FUNCTION_BLOCK FB_Estacion
VAR_INPUT
	// SFC-Flags
	SFCReset: BOOL;
	
	// Parámetros
	TpoEstabilidad: TIME := T#1000MS;
	UdsSolicitadas:UINT := 5;
	
END_VAR
VAR_OUTPUT
	// Parámetros
	CondicionInicial: BOOL;
	UdsPendientes: UINT;
	UdsRealizadas: BOOL;
	
	// Entradas comunes
	PulsadorEmergencia AT %I*: BOOL;
    SelectorManual AT %I*: BOOL;
    PulsadorMarcha AT %I*: BOOL;
    PulsadorParada AT %I*: BOOL := TRUE; // Contacto normalmente cerrado
    EstacionConectada AT %I*: BOOL := TRUE;
    DetectorPresion AT %I*: BOOL := TRUE;
	
	PalePresencia AT %I*: BOOL;
    PaleCodigoBit0 AT %I*: BOOL;
    PaleCodigoBit1 AT %I*: BOOL;
    PaleCodigoBit2 AT %I*: BOOL;
	
	// Entradas específicas
	DescargadorDetras AT %I*: BOOL;
	DescargadorDelante AT %I*: BOOL;
	VerticalArriba AT %I*: BOOL;
	VerticalAbajo AT %I*: BOOL;
	VerificadorArriba AT %I*: BOOL;
	VerificadorAbajo AT %I*: BOOL;
	DesplazadorDetras AT %I*: BOOL;
	AlimentadorDetras AT %I*: BOOL;
	AlimentadorDelante AT %I*: BOOL;
	VacioDescargador AT %I*: BOOL;
	PresenciaBaseAlimentador AT %I*:BOOL;
END_VAR
VAR
	// Bloques funcionales
	CLK: FB_Clock;
	// Salidas comunes
	DesconectaEstacion AT %Q*: BOOL;
    LamparaAlarma AT %Q*: BOOL;
    LamparaMarcha AT %Q*: BOOL;
	LamparaFaltaMaterial AT %Q*: BOOL;
    AvisadorSonoro AT %Q*: BOOL;

    CintaMotorActiva AT %Q*: BOOL;
    CintaMotorInvierte AT %Q*: BOOL;
    CintaRetenedorBaja AT %Q*: BOOL;
    CintaSeparadorSube AT %Q*: BOOL;
	
	// Salidas específicas
	DescargadorAtras AT %Q*: BOOL;
	DescargadorAdelante AT %Q*: BOOL;
	DescargadorBaja AT %Q*: BOOL;
	RechazadorAdelante AT %Q*: BOOL;
	VerificadorBaja AT %Q*: BOOL;
	DesplazadorAdelante AT %Q*: BOOL;
	AlimentadorAdelante AT %Q*: BOOL;
	EyectorSucciona AT %Q*: BOOL;
END_VAR

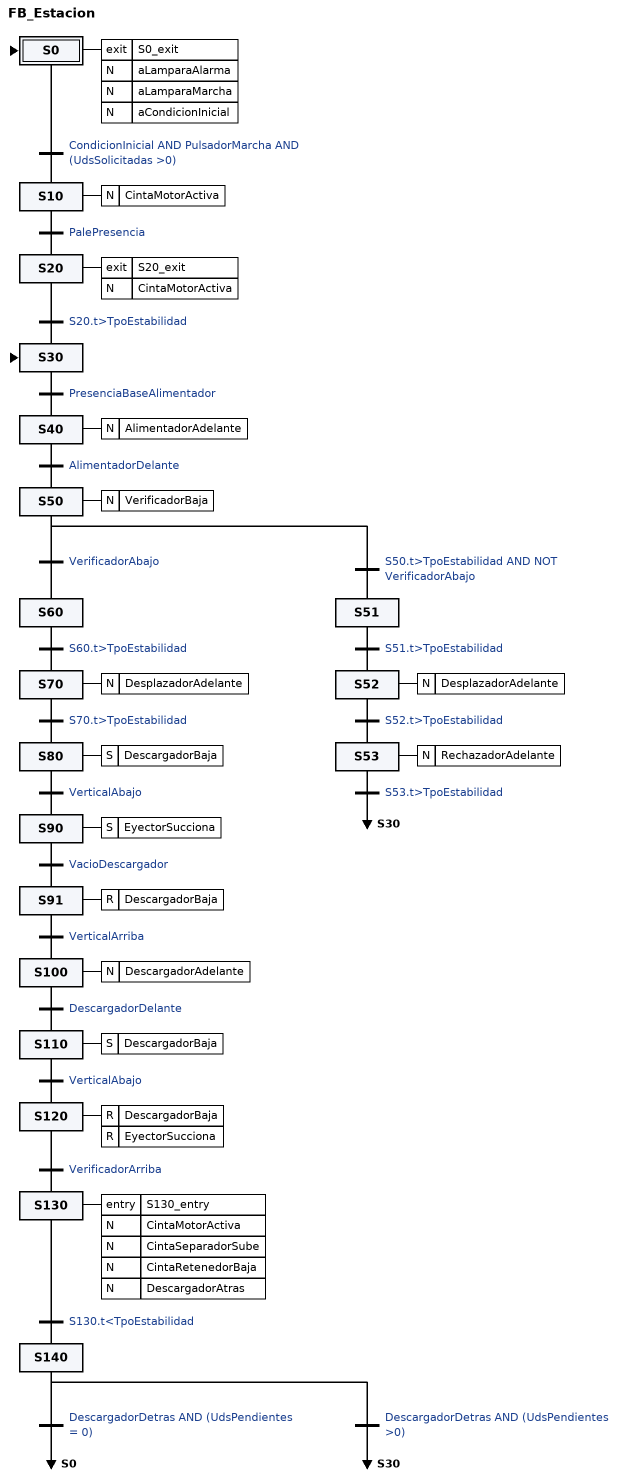
INITIAL_STEP S0:
    S0_exit(P0);  // exit action
    aLamparaAlarma(N);
    aLamparaMarcha(N);
    aCondicionInicial(N);
END_STEP
TRANSITION FROM S0 TO S10
    := CondicionInicial AND PulsadorMarcha AND (UdsSolicitadas >0);
END_TRANSITION
STEP S10:
    CintaMotorActiva(N);
END_STEP
TRANSITION FROM S10 TO S20
    := PalePresencia;
END_TRANSITION
STEP S20:
    S20_exit(P0);  // exit action
    CintaMotorActiva(N);
END_STEP
TRANSITION FROM S20 TO S30
    := S20.t>TpoEstabilidad;
END_TRANSITION
STEP S30:
END_STEP
TRANSITION FROM S30 TO S40
    := PresenciaBaseAlimentador;
END_TRANSITION
STEP S40:
    AlimentadorAdelante(N);
END_STEP
TRANSITION FROM S40 TO S50
    := AlimentadorDelante;
END_TRANSITION
STEP S50:
    VerificadorBaja(N);
END_STEP
TRANSITION FROM S50 TO S60
    := VerificadorAbajo;
END_TRANSITION
TRANSITION FROM S50 TO S51
    := S50.t>TpoEstabilidad AND NOT VerificadorAbajo;
END_TRANSITION
STEP S51:
END_STEP
TRANSITION FROM S51 TO S52
    := S51.t>TpoEstabilidad;
END_TRANSITION
STEP S52:
    DesplazadorAdelante(N);
END_STEP
TRANSITION FROM S52 TO S53
    := S52.t>TpoEstabilidad;
END_TRANSITION
STEP S53:
    RechazadorAdelante(N);
END_STEP
TRANSITION FROM S53 TO S30
    := S53.t>TpoEstabilidad;
END_TRANSITION
STEP S60:
END_STEP
TRANSITION FROM S60 TO S70
    := S60.t>TpoEstabilidad;
END_TRANSITION
STEP S70:
    DesplazadorAdelante(N);
END_STEP
TRANSITION FROM S70 TO S80
    := S70.t>TpoEstabilidad;
END_TRANSITION
STEP S80:
    DescargadorBaja(S);
END_STEP
TRANSITION FROM S80 TO S90
    := VerticalAbajo;
END_TRANSITION
STEP S90:
    EyectorSucciona(S);
END_STEP
TRANSITION FROM S90 TO S91
    := VacioDescargador;
END_TRANSITION
STEP S91:
    DescargadorBaja(R);
END_STEP
TRANSITION FROM S91 TO S100
    := VerticalArriba;
END_TRANSITION
STEP S100:
    DescargadorAdelante(N);
END_STEP
TRANSITION FROM S100 TO S110
    := DescargadorDelante;
END_TRANSITION
STEP S110:
    DescargadorBaja(S);
END_STEP
TRANSITION FROM S110 TO S120
    := VerticalAbajo;
END_TRANSITION
STEP S120:
    DescargadorBaja(R);
    EyectorSucciona(R);
END_STEP
TRANSITION FROM S120 TO S130
    := VerificadorArriba;
END_TRANSITION
STEP S130:
    S130_entry(P1);  // entry action
    CintaMotorActiva(N);
    CintaSeparadorSube(N);
    CintaRetenedorBaja(N);
    DescargadorAtras(N);
END_STEP
TRANSITION FROM S130 TO S140
    := S130.t<TpoEstabilidad;
END_TRANSITION
STEP S140:
END_STEP
TRANSITION FROM S140 TO S0
    := DescargadorDetras AND (UdsPendientes = 0);
END_TRANSITION
TRANSITION FROM S140 TO S30
    := DescargadorDetras AND (UdsPendientes >0);
END_TRANSITION

ACTION aCondicionInicial:
CondicionInicial:= EstacionConectada AND AlimentadorDetras AND DesplazadorDetras  AND VerificadorArriba AND DescargadorDetras;
END_ACTION

ACTION aLamparaAlarma:
LamparaAlarma := (S0.x AND NOT CondicionInicial AND CLK.Q);
END_ACTION

ACTION aLamparaMarcha:
LamparaMarcha := (S0.x AND CondicionInicial AND CLK.Q) OR NOT S0.x;

CLK();
END_ACTION

ACTION aPaleCodigo:
PaleCodigoBit0.0 := PaleCodigoBit0;
PaleCodigoBit0.1 := PaleCodigoBit1;
PaleCogidoBit1.2 := PaleCodigoBit2;
END_ACTION

ACTION S0_exit:
// Actualizamos el número de uds cada vez que se inicia
IF (UdsPendientes = 0) THEN
	UdsPendientes := UdsSolicitadas;
END_IF
END_ACTION

ACTION S130_entry:
// Al completar correctamente la transferencia
// Actualizamos el número de unidades realizadas
UdsRealizadas := UdsRealizadas + 1;

// Si quedan unidades pendientes actualizamos también su valor
IF (UdsPendientes >0) THEN
	UdsPendientes := UdsPendientes -1;
END_IF
END_ACTION

ACTION S20_exit:
aPaleCodigo();
END_ACTION

END_FUNCTION_BLOCK

(* stored: Version 1.1.0.1, ProductVersion 3.1.4024.12
   POU FB_Estacion: Id {5e144844-4386-40ba-949a-26810c81a1f5}, SpecialFunc None
   Action aCondicionInicial: Id {bf32252c-e507-4d44-952e-8305a32926c4}
   Action aLamparaAlarma: Id {cac2a3fa-3003-4214-9d5a-6c08083911e3}
   Action aLamparaMarcha: Id {94b12d36-447f-436c-a948-a622a2fc9f4a}
   Action aPaleCodigo: Id {39e77257-dc52-4484-8645-6cb060f90db9}
   Action S0_exit: Id {39489810-d099-4953-8ff2-1b94001cab29}
   Action S130_entry: Id {f406c43e-c925-4b32-b1a4-adf31d5fc15d}
   Action S20_exit: Id {630d9ff6-7226-4e79-9971-3c2d10d66ba8} *)
